# EPICS substitutions: iocBoot/iocSoftGlue/softGlue_FPGAContentDev.substitutions
file "$(SOFTGLUE)/softGlueApp/Db/softGlue_Input.db"
{
pattern {P  H 	SIG					PORT	ADDR}

{xxx: softGlue: AND-1_IN1			SOFTGLUE 0x8000B0}
{xxx: softGlue: AND-1_IN2			SOFTGLUE 0x8000B8}

{xxx: softGlue: AND-2_IN1			SOFTGLUE 0x8000D0}
{xxx: softGlue: AND-2_IN2			SOFTGLUE 0x8000D8}

{xxx: softGlue: OR-1_IN1			SOFTGLUE 0x8000F0}
{xxx: softGlue: OR-1_IN2			SOFTGLUE 0x8000F8}

{xxx: softGlue: OR-2_IN1			SOFTGLUE 0x800110}
{xxx: softGlue: OR-2_IN2			SOFTGLUE 0x800118}

{xxx: softGlue: XOR-1_IN1			SOFTGLUE 0x800130}
{xxx: softGlue: XOR-1_IN2			SOFTGLUE 0x800138}

{xxx: softGlue: XOR-2_IN1			SOFTGLUE 0x800150}
{xxx: softGlue: XOR-2_IN2			SOFTGLUE 0x800158}

{xxx: softGlue: DEMUX2-1_IN			SOFTGLUE 0x800170}
{xxx: softGlue: DEMUX2-1_SEL		SOFTGLUE 0x800178}

{xxx: softGlue: DEMUX2-2_IN			SOFTGLUE 0x800190}
{xxx: softGlue: DEMUX2-2_SEL		SOFTGLUE 0x800198}

{xxx: softGlue: DFF-1_D				SOFTGLUE 0x800270}
{xxx: softGlue: DFF-1_CLOCK			SOFTGLUE 0x800278}
{xxx: softGlue: DFF-1_SET			SOFTGLUE 0x800280}
{xxx: softGlue: DFF-1_CLEAR			SOFTGLUE 0x800288}

{xxx: softGlue: DFF-2_D				SOFTGLUE 0x8002A0}
{xxx: softGlue: DFF-2_CLOCK			SOFTGLUE 0x8002A8}
{xxx: softGlue: DFF-2_SET			SOFTGLUE 0x8002B0}
{xxx: softGlue: DFF-2_CLEAR			SOFTGLUE 0x8002B8}

{xxx: softGlue: DivByN-1_ENABLE		SOFTGLUE 0x8001e0}
{xxx: softGlue: DivByN-1_CLOCK		SOFTGLUE 0x8001e8}
{xxx: softGlue: DivByN-1_RESET		SOFTGLUE 0x8001f0}

{xxx: softGlue: DivByN-2_ENABLE		SOFTGLUE 0x800240}
{xxx: softGlue: DivByN-2_CLOCK		SOFTGLUE 0x800248}
{xxx: softGlue: DivByN-2_RESET		SOFTGLUE 0x800250}

{xxx: softGlue: DnCntr-1_ENABLE		SOFTGLUE 0x8001B8}
{xxx: softGlue: DnCntr-1_CLOCK		SOFTGLUE 0x8001B0}
{xxx: softGlue: DnCntr-1_LOAD		SOFTGLUE 0x8001C0}

{xxx: softGlue: DnCntr-2_ENABLE		SOFTGLUE 0x800218}
{xxx: softGlue: DnCntr-2_CLOCK		SOFTGLUE 0x800210}
{xxx: softGlue: DnCntr-2_LOAD		SOFTGLUE 0x800220}

{xxx: softGlue: MUX2-1_IN0			SOFTGLUE 0x8002D0}
{xxx: softGlue: MUX2-1_IN1			SOFTGLUE 0x8002D8}
{xxx: softGlue: MUX2-1_SEL			SOFTGLUE 0x8002E0}

{xxx: softGlue: MUX2-2_IN0			SOFTGLUE 0x8002F0}
{xxx: softGlue: MUX2-2_IN1			SOFTGLUE 0x8002F8}
{xxx: softGlue: MUX2-2_SEL			SOFTGLUE 0x800300}

{xxx: softGlue: UpCntr-1_ENABLE		SOFTGLUE 0x800318}
{xxx: softGlue: UpCntr-1_CLOCK		SOFTGLUE 0x800310}
{xxx: softGlue: UpCntr-1_CLEAR		SOFTGLUE 0x800320}

{xxx: softGlue: UpCntr-2_ENABLE		SOFTGLUE 0x800338}
{xxx: softGlue: UpCntr-2_CLOCK		SOFTGLUE 0x800330}
{xxx: softGlue: UpCntr-2_CLEAR		SOFTGLUE 0x800340}

# These are outputs from the user's viewpoint, but they behave like softGlue
# inputs.
{xxx: softGlue: FO1					SOFTGLUE 0x800070}
{xxx: softGlue: FO2					SOFTGLUE 0x800078}
{xxx: softGlue: FO3					SOFTGLUE 0x800080}
{xxx: softGlue: FO4					SOFTGLUE 0x800088}
{xxx: softGlue: FO5					SOFTGLUE 0x800090}
{xxx: softGlue: FO6					SOFTGLUE 0x800098}
{xxx: softGlue: FO7					SOFTGLUE 0x8000A0}
{xxx: softGlue: FO8					SOFTGLUE 0x8000A8}
{xxx: softGlue: FO9					SOFTGLUE 0x800390}
{xxx: softGlue: FO10				SOFTGLUE 0x800398}
{xxx: softGlue: FO11				SOFTGLUE 0x8003A0}
{xxx: softGlue: FO12				SOFTGLUE 0x8003A8}
{xxx: softGlue: FO13				SOFTGLUE 0x8003B0}
{xxx: softGlue: FO14				SOFTGLUE 0x8003B8}
{xxx: softGlue: FO15				SOFTGLUE 0x8003C0}
{xxx: softGlue: FO16				SOFTGLUE 0x8003C8}
}

file "$(SOFTGLUE)/softGlueApp/Db/softGlue_Output.db"
{
pattern {P  H 	SIG					PORT	ADDR}

{xxx: softGlue: AND-1_POUT			SOFTGLUE 0x8000C0}
{xxx: softGlue: AND-1_NOUT			SOFTGLUE 0x8000C8}

{xxx: softGlue: AND-2_POUT			SOFTGLUE 0x8000E0}
{xxx: softGlue: AND-2_NOUT			SOFTGLUE 0x8000E8}

{xxx: softGlue: OR-1_POUT			SOFTGLUE 0x800100}
{xxx: softGlue: OR-1_NOUT			SOFTGLUE 0x800108}

{xxx: softGlue: OR-2_POUT			SOFTGLUE 0x800120}
{xxx: softGlue: OR-2_NOUT			SOFTGLUE 0x800128}

{xxx: softGlue: XOR-1_POUT			SOFTGLUE 0x800140}
{xxx: softGlue: XOR-1_NOUT			SOFTGLUE 0x800148}

{xxx: softGlue: XOR-2_POUT			SOFTGLUE 0x800160}
{xxx: softGlue: XOR-2_NOUT			SOFTGLUE 0x800168}

{xxx: softGlue: DEMUX2-1_OUT0		SOFTGLUE 0x800180}
{xxx: softGlue: DEMUX2-1_OUT1		SOFTGLUE 0x800188}

{xxx: softGlue: DEMUX2-2_OUT0		SOFTGLUE 0x8001A0}
{xxx: softGlue: DEMUX2-2_OUT1		SOFTGLUE 0x8001A8}

{xxx: softGlue: DFF-1_POUT			SOFTGLUE 0x800290}
{xxx: softGlue: DFF-1_NOUT			SOFTGLUE 0x800298}

{xxx: softGlue: DFF-2_POUT			SOFTGLUE 0x8002C0}
{xxx: softGlue: DFF-2_NOUT			SOFTGLUE 0x8002C8}

{xxx: softGlue: DivByN-1_POUT		SOFTGLUE 0x8001f8}
{xxx: softGlue: DivByN-1_NOUT		SOFTGLUE 0x800200}

{xxx: softGlue: DivByN-2_POUT		SOFTGLUE 0x800258}
{xxx: softGlue: DivByN-2_NOUT		SOFTGLUE 0x800260}

{xxx: softGlue: DnCntr-1_POUT		SOFTGLUE 0x8001C8}
{xxx: softGlue: DnCntr-1_NOUT		SOFTGLUE 0x8001D0}

{xxx: softGlue: DnCntr-2_POUT		SOFTGLUE 0x800228}
{xxx: softGlue: DnCntr-2_NOUT		SOFTGLUE 0x800230}

{xxx: softGlue: MUX2-1_OUT			SOFTGLUE 0x8002E8}
{xxx: softGlue: MUX2-2_OUT			SOFTGLUE 0x800308}

{xxx: softGlue: 8MHZ_CLK			SOFTGLUE 0x8003E0}

# These are inputs from the user's viewpoint, but they behave like softGlue
# outputs.
{xxx: softGlue: FI1					SOFTGLUE 0x800030}
{xxx: softGlue: FI2					SOFTGLUE 0x800038}
{xxx: softGlue: FI3					SOFTGLUE 0x800040}
{xxx: softGlue: FI4					SOFTGLUE 0x800048}
{xxx: softGlue: FI5					SOFTGLUE 0x800050}
{xxx: softGlue: FI6					SOFTGLUE 0x800058}
{xxx: softGlue: FI7					SOFTGLUE 0x800060}
{xxx: softGlue: FI8					SOFTGLUE 0x800068}
{xxx: softGlue: FI9					SOFTGLUE 0x800350}
{xxx: softGlue: FI10				SOFTGLUE 0x800358}
{xxx: softGlue: FI11				SOFTGLUE 0x800360}
{xxx: softGlue: FI12				SOFTGLUE 0x800368}
{xxx: softGlue: FI13				SOFTGLUE 0x800370}
{xxx: softGlue: FI14				SOFTGLUE 0x800378}
{xxx: softGlue: FI15				SOFTGLUE 0x800380}
{xxx: softGlue: FI16				SOFTGLUE 0x800388}
}

file "$(SOFTGLUE)/softGlueApp/Db/softGlue_Register.db"
{
pattern {P  H 	SIG					PORT	ADDR	CALC}

{xxx: softGlue: DnCntr-1_PRESET		SOFTGLUE 0x8001D8	A-1}
{xxx: softGlue: DnCntr-2_PRESET		SOFTGLUE 0x800238	A-1}

{xxx: softGlue: DivByN-1_N			SOFTGLUE 0x800208	A-1}
{xxx: softGlue: DivByN-2_N			SOFTGLUE 0x800268	A-1}

}

file "$(SOFTGLUE)/softGlueApp/Db/softGlue_InRegister32.db"
{
pattern {P  H 	SIG					PORT		ADDR_MSW ADDR_LSW}

{xxx: softGlue: UpCntr-1_COUNTS		SOFTGLUE	0x8003D0 0x800328}
{xxx: softGlue: UpCntr-2_COUNTS		SOFTGLUE	0x8003D8 0x800348}
}
